Omron CX-Programmer project NewProject (CX-Programmer 9.61)

# PLC NewPLC1: CP1H XA

## Global symbols (name address type ; comment)
0.00 BOOL  ; F1LSw
0.01 BOOL  ; F2LSw
0.02 BOOL  ; F3LSw
0.03 BOOL  ; F1CC
0.04 BOOL  ; F1HCUp
0.05 BOOL  ; F2CC
0.06 BOOL  ; F2HCUp
0.07 BOOL  ; F2HCDown
0.08 BOOL  ; F3CC
0.09 BOOL  ; F3HCDown
0.10 BOOL  ; F1SlowL
0.11 BOOL  ; F2SlowL
0.12 BOOL  ; F3SlowL
0.13 BOOL  ; ManualDoorOpen
100.00 BOOL  ; L1
100.01 BOOL  ; L2
100.02 BOOL  ; L3
100.03 BOOL  ; A1
100.04 BOOL  ; A2
100.05 BOOL  ; A3
100.06 BOOL  ; Stop
100.07 BOOL  ; Memory1ForVisit
100.08 BOOL  ; Memory2ForVisit
100.09 BOOL  ; LS1
100.10 BOOL  ; LS2
100.11 BOOL  ; LS3
100.12 BOOL  ; SM
100.13 BOOL  ; DO
100.14 BOOL  ; UpM
100.15 BOOL  ; DownM
101.00 BOOL  ; M1
101.01 BOOL  ; M2
10.00 BOOL  ; OpenDoor
10.01 BOOL  ; Up
10.02 BOOL  ; Down
10.03 BOOL  ; Slow
1.00 BOOL  ; SystemStart
1.01 BOOL  ; SystemStop
1.03 BOOL  ; F1HCUp
T0000 BOOL  ; Timer1
T0001 BOOL  ; Timer2
T0002 BOOL  ; Timer3

## Program NewProgram1 (cyclic task 0)

### Section Section1

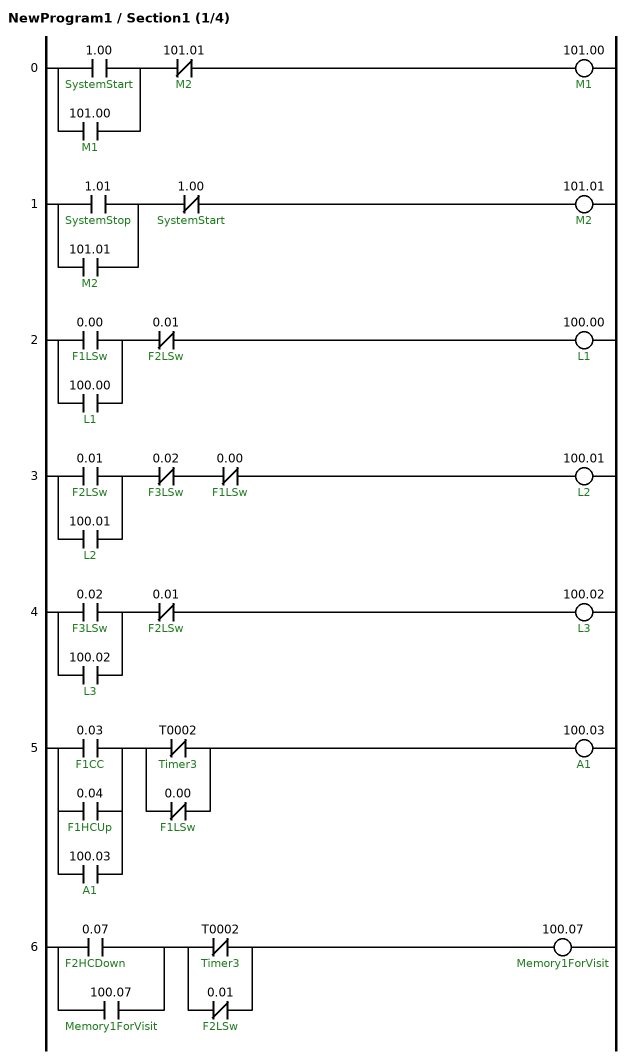
; rung 0
LD 1.00  ; SystemStart
OR 101.00  ; M1
ANDNOT 101.01  ; M2
OUT 101.00  ; M1
; rung 1
LD 1.01  ; SystemStop
OR 101.01  ; M2
ANDNOT 1.00  ; SystemStart
OUT 101.01  ; M2
; rung 2
LD 0.00  ; F1LSw
OR 100.00  ; L1
ANDNOT 0.01  ; F2LSw
OUT 100.00  ; L1
; rung 3
LD 0.01  ; F2LSw
OR 100.01  ; L2
ANDNOT 0.02  ; F3LSw
ANDNOT 0.00  ; F1LSw
OUT 100.01  ; L2
; rung 4
LD 0.02  ; F3LSw
OR 100.02  ; L3
ANDNOT 0.01  ; F2LSw
OUT 100.02  ; L3
; rung 5
LD 0.03  ; F1CC
OR 0.04  ; F1HCUp
OR 100.03  ; A1
LDNOT T0002  ; Timer3
ORNOT 0.00  ; F1LSw
ANDLD
OUT 100.03  ; A1
; rung 6
LD 0.07  ; F2HCDown
OR 100.07  ; Memory1ForVisit
LDNOT T0002  ; Timer3
ORNOT 0.01  ; F2LSw
ANDLD
OUT 100.07  ; Memory1ForVisit

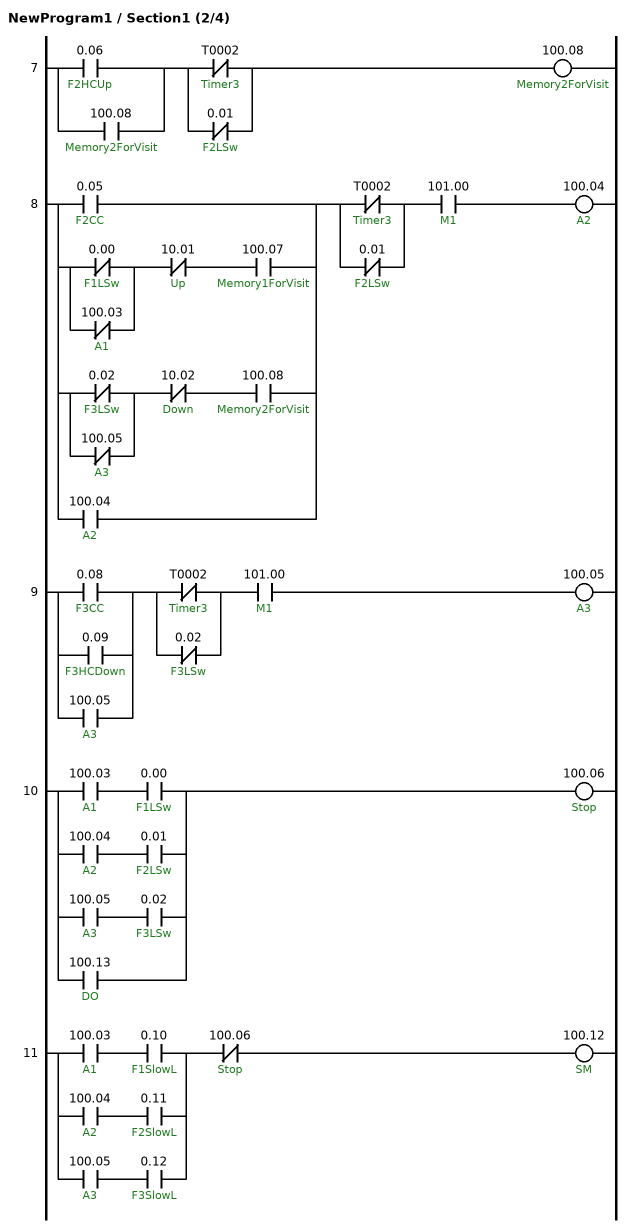
; rung 7
LD 0.06  ; F2HCUp
OR 100.08  ; Memory2ForVisit
LDNOT T0002  ; Timer3
ORNOT 0.01  ; F2LSw
ANDLD
OUT 100.08  ; Memory2ForVisit
; rung 8
LD 0.05  ; F2CC
LDNOT 0.00  ; F1LSw
ORNOT 100.03  ; A1
ANDNOT 10.01  ; Up
AND 100.07  ; Memory1ForVisit
ORLD
LDNOT 0.02  ; F3LSw
ORNOT 100.05  ; A3
ANDNOT 10.02  ; Down
AND 100.08  ; Memory2ForVisit
ORLD
OR 100.04  ; A2
LDNOT T0002  ; Timer3
ORNOT 0.01  ; F2LSw
ANDLD
AND 101.00  ; M1
OUT 100.04  ; A2
; rung 9
LD 0.08  ; F3CC
OR 0.09  ; F3HCDown
OR 100.05  ; A3
LDNOT T0002  ; Timer3
ORNOT 0.02  ; F3LSw
ANDLD
AND 101.00  ; M1
OUT 100.05  ; A3
; rung 10
LD 100.03  ; A1
AND 0.00  ; F1LSw
LD 100.04  ; A2
AND 0.01  ; F2LSw
ORLD
LD 100.05  ; A3
AND 0.02  ; F3LSw
ORLD
OR 100.13  ; DO
OUT 100.06  ; Stop
; rung 11
LD 100.03  ; A1
AND 0.10  ; F1SlowL
LD 100.04  ; A2
AND 0.11  ; F2SlowL
ORLD
LD 100.05  ; A3
AND 0.12  ; F3SlowL
ORLD
ANDNOT 100.06  ; Stop
OUT 100.12  ; SM

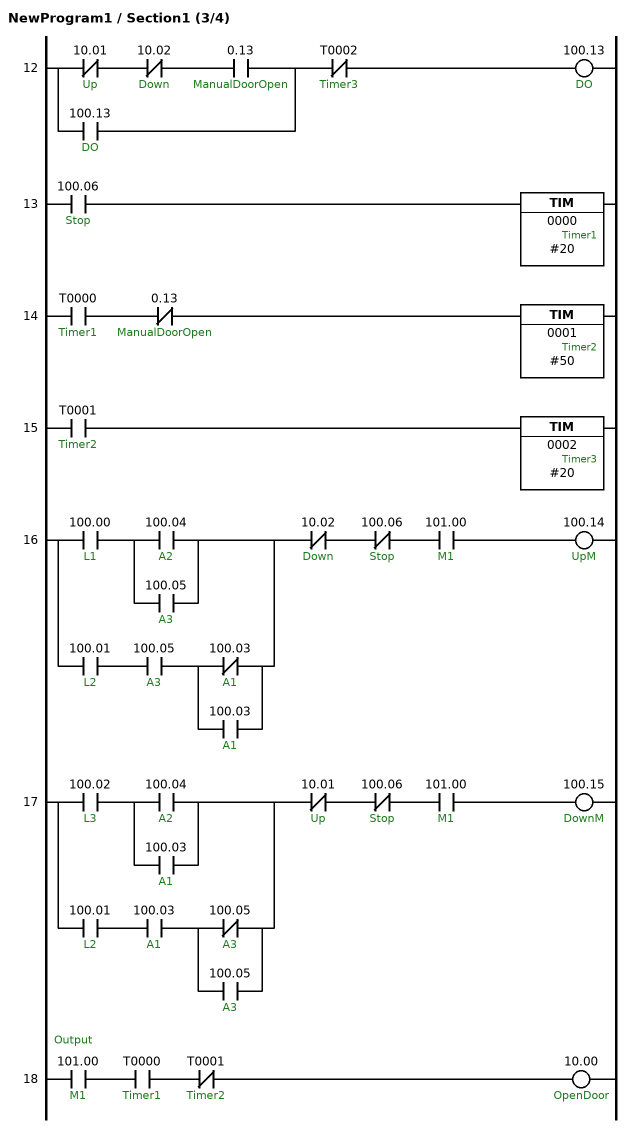
; rung 12
LDNOT 10.01  ; Up
ANDNOT 10.02  ; Down
AND 0.13  ; ManualDoorOpen
OR 100.13  ; DO
ANDNOT T0002  ; Timer3
OUT 100.13  ; DO
; rung 13
LD 100.06  ; Stop
TIM 0000 #20  ; Timer1
; rung 14
LD T0000  ; Timer1
ANDNOT 0.13  ; ManualDoorOpen
TIM 0001 #50  ; Timer2
; rung 15
LD T0001  ; Timer2
TIM 0002 #20  ; Timer3
; rung 16
LD 100.00  ; L1
LD 100.04  ; A2
OR 100.05  ; A3
ANDLD
LD 100.01  ; L2
AND 100.05  ; A3
LDNOT 100.03  ; A1
OR 100.03  ; A1
ANDLD
ORLD
ANDNOT 10.02  ; Down
ANDNOT 100.06  ; Stop
AND 101.00  ; M1
OUT 100.14  ; UpM
; rung 17
LD 100.02  ; L3
LD 100.04  ; A2
OR 100.03  ; A1
ANDLD
LD 100.01  ; L2
AND 100.03  ; A1
LDNOT 100.05  ; A3
OR 100.05  ; A3
ANDLD
ORLD
ANDNOT 10.01  ; Up
ANDNOT 100.06  ; Stop
AND 101.00  ; M1
OUT 100.15  ; DownM
; rung 18: Output
LD 101.00  ; M1
AND T0000  ; Timer1
ANDNOT T0001  ; Timer2
OUT 10.00  ; OpenDoor

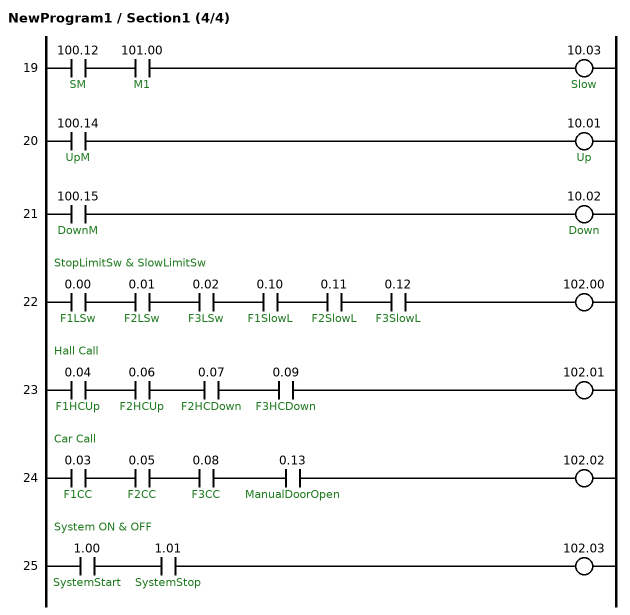
; rung 19
LD 100.12  ; SM
AND 101.00  ; M1
OUT 10.03  ; Slow
; rung 20
LD 100.14  ; UpM
OUT 10.01  ; Up
; rung 21
LD 100.15  ; DownM
OUT 10.02  ; Down
; rung 22: StopLimitSw & SlowLimitSw
LD 0.00  ; F1LSw
AND 0.01  ; F2LSw
AND 0.02  ; F3LSw
AND 0.10  ; F1SlowL
AND 0.11  ; F2SlowL
AND 0.12  ; F3SlowL
OUT 102.00
; rung 23: Hall Call
LD 0.04  ; F1HCUp
AND 0.06  ; F2HCUp
AND 0.07  ; F2HCDown
AND 0.09  ; F3HCDown
OUT 102.01
; rung 24: Car Call
LD 0.03  ; F1CC
AND 0.05  ; F2CC
AND 0.08  ; F3CC
AND 0.13  ; ManualDoorOpen
OUT 102.02
; rung 25: System ON & OFF
LD 1.00  ; SystemStart
AND 1.01  ; SystemStop
OUT 102.03

### Section END
; rung 0
END(001)